TYPE T_OAC_Filename : T_MaxString;
END_TYPE

(* stored: Version 1.1.0.1
   DUT T_OAC_Filename: Id {bb11b787-8967-4a47-aa69-13e10e414b26} *)
